{attribute 'linkalways'} 
{attribute 'no_explicit_call' := 'This FB is a CLASS and must be accessed using methods or properties'}
{attribute 'enable_dynamic_creation'}
FUNCTION_BLOCK Node_F_VN_ContourOrientation EXTENDS VisionNode
VAR
    ipContour : _ITcVnContainer;
    stOrientation : _TcVnRotatedRectangle;
    hrPrev : _HRESULT(S_OK);
	hresult : _HRESULT(S_OK);
END_VAR

METHOD PUBLIC  Clone : I_Node
VAR
	pNode : POINTER TO Node_F_VN_ContourOrientation;
END_VAR
pNode := __NEW(Node_F_VN_ContourOrientation);
Clone := pNode^;
END_METHOD

METHOD FB_init : BOOL
VAR_INPUT
	bInitRetains : BOOL; // if TRUE, the retain variables are initialized (warm start / cold start)
	bInCopyCode : BOOL;  // if TRUE, the instance afterwards gets moved into the copy code (online change)
END_VAR
AddInput('ipContour', ipContour);
AddInput('hrPrev', hrPrev);
AddOutput('stOrientation', stOrientation);
AddOutput('hresult',hresult);
END_METHOD

METHOD PROTECTED OnExecute
hresult.Value := F_VN_ContourOrientation(
	ipContour := ipContour.Value,
    stOrientation := stOrientation.Value,
	hrPrev:= hrPrev.Value);
END_METHOD

METHOD PUBLIC PreExecutionCheck
VAR_INPUT
	Check : I_PreExecutionChecks;
END_VAR
Check.IsTrue(ipContour.IsValid, 'ipContour must be a valid container');
Check.IsTrue((ipContour.IsType(TC_GLOBAL_CONST_LIST.ContainerType_Vector_TcVnPoint2_DINT) OR
              ipContour.IsType(TC_GLOBAL_CONST_LIST.ContainerType_Vector_TcVnPoint2_REAL) OR
              ipContour.IsType(TC_GLOBAL_CONST_LIST.ContainerType_Vector_TcVnPoint2_LREAL)),
              'ipContour contains incorrect type');
END_METHOD

END_FUNCTION_BLOCK

(* stored: Version 1.1.0.1, ProductVersion 3.1.4026.13
   POU Node_F_VN_ContourOrientation: Id {2df0dd1e-0b78-0ccf-265b-335876f2f1b6}, SpecialFunc None
   Folder Constructor: Id {f7d18d9c-c40d-0834-32a2-8c7ff08e3004}
   Method Clone: Id {01ed077c-f375-0a97-1ad6-502ad584a133}
   Method FB_init: Id {e38391fe-11b9-0dcc-03c0-4b04a3e146eb}
   Method OnExecute: Id {5b78fbcd-1d3d-0723-27da-d6d18f83ed48}
   Method PreExecutionCheck: Id {fb662b89-5b03-099a-29c9-5486c1263389} *)
